// TwinCAT 3 PLC project Sample02
// ProgramVersion: 3.1.4020.10
// libraries:
//   Tc2_Standard, * (Beckhoff Automation GmbH)
//   Tc2_System, * (Beckhoff Automation GmbH)
//   Tc3_Module, * (Beckhoff Automation GmbH)
// project tree:
//   / PlcTask.TcTTO (not stored)
//   POUs/Commands/ FB_AirConComfortCommand.TcPOU (not stored), FB_AirConStandbyCommand.TcPOU (not stored), FB_LampSetLevelCommand.TcPOU (not stored), FB_MusicPlayCommand.TcPOU (not stored), FB_MusicStopCommand.TcPOU (not stored), FB_RoomOffCommand.TcPOU (not stored), FB_SocketOffCommand.TcPOU (not stored), FB_SocketOnCommand.TcPOU (not stored), I_Command.TcIO (not stored)
//   POUs/Invoker/ FB_SwitchPanel.TcPOU (not stored)
//   POUs/ MAIN.TcPOU
//   POUs/Receiver/ FB_AirConditioning.TcPOU (not stored), FB_CDPlayer.TcPOU (not stored), FB_Lamp.TcPOU (not stored), FB_Socket.TcPOU (not stored)
// real-time tasks:
//   TASK PlcTask: cycle T#10ms, priority 20, ADS port 350

// ---- POUs/MAIN.TcPOU
PROGRAM MAIN
VAR
	// Invoker
	fbSwitchPanel				: FB_SwitchPanel;
	
	// Receiver
	fbSocket					: FB_Socket;
	refSocket					: REFERENCE TO FB_Socket := fbSocket;	
	fbLamp						: FB_Lamp;
	refLamp						: REFERENCE TO FB_Lamp := fbLamp;	
	fbAirConditioning			: FB_AirConditioning;
	refAirConditioning			: REFERENCE TO FB_AirConditioning := fbAirConditioning;
	fbCDPlayer					: FB_CDPlayer;
	refCDPlayer					: REFERENCE TO FB_CDPlayer := fbCDPlayer;

	// Commands
	fbSocketOnCommand			: FB_SocketOnCommand(refSocket);
	fbSocketOffCommand			: FB_SocketOffCommand(refSocket);
	fbLampSetLevel100Command	: FB_LampSetLevelCommand(refLamp, 100);
	fbLampSetLevel0Command		: FB_LampSetLevelCommand(refLamp, 0);
	fbAirConComfortCommand		: FB_AirConComfortCommand(refAirConditioning);
	fbAirConStandbyCommand		: FB_AirConStandbyCommand(refAirConditioning);	
	fbMusicPlayCommand			: FB_MusicPlayCommand(refCDPlayer);
	fbMusicStopCommand			: FB_MusicStopCommand(refCDPlayer);	
	fbRoomOffCommand			: FB_RoomOffCommand(fbSocketOffCommand, fbLampSetLevel0Command, fbAirConStandbyCommand, fbMusicStopCommand);	
	bInit						: BOOL;
END_VAR

IF (NOT bInit) THEN
	fbSwitchPanel.SetCommand(1, fbSocketOnCommand);
	fbSwitchPanel.SetCommand(2, fbSocketOffCommand);
	fbSwitchPanel.SetCommand(3, fbLampSetLevel100Command);
	fbSwitchPanel.SetCommand(4, fbLampSetLevel0Command);
	fbSwitchPanel.SetCommand(5, fbAirConComfortCommand);
	fbSwitchPanel.SetCommand(6, fbAirConStandbyCommand);
	fbSwitchPanel.SetCommand(7, fbMusicPlayCommand);
	fbSwitchPanel.SetCommand(8, fbRoomOffCommand);
	bInit := TRUE;
ELSE
	fbSwitchPanel();	
END_IF

END_PROGRAM
